INTERFACE I_NodeFactory

METHOD PUBLIC Accept
VAR_INPUT
	Visitor : I_NodeFactoryVisitor;
END_VAR
END_METHOD

METHOD AddNodeAsPrototype : I_NodePrototype
VAR_INPUT
	Path : T_MAXSTRING;
	Node : I_Node;
END_VAR
END_METHOD

METHOD PUBLIC AddNodePrototype
VAR_INPUT
	NodePrototype : I_NodePrototype;
END_VAR
END_METHOD

METHOD PUBLIC InstallNodePack
VAR_INPUT
	NodePack : I_NodePack;
END_VAR
END_METHOD

PROPERTY PUBLIC ABSTRACT NodePrototypes : I_NodePrototypes
GET
END_GET
END_PROPERTY

METHOD PUBLIC TryCreateNodeByType : BOOL
VAR_INPUT
	Path : T_MAXSTRING;
	Destination : REFERENCE TO I_Node;
END_VAR
END_METHOD

END_INTERFACE

(* stored: Version 1.1.0.1, ProductVersion 3.1.4024.12
   Itf I_NodeFactory: Id {1c91137c-0d76-4a0b-982f-ff1013ab557c}
   Method Accept: Id {f6a58bad-0d11-4651-b4e3-e6b638da37c0}
   Method AddNodeAsPrototype: Id {3c290acf-ef58-4296-9f99-efa7638f18a5}
   Method AddNodePrototype: Id {fca90214-0e16-4176-8cb8-b68284861d51}
   Method InstallNodePack: Id {eeb92a5b-c90e-441b-8a57-23a935768eb2}
   Property NodePrototypes: Id {82e304d3-cf5f-4e21-8935-71cbe599f257}
   Get Get: Id {4cb802dd-fdb8-4d8d-8602-1230b292a15c}
   Method TryCreateNodeByType: Id {c6542a73-8c2a-431b-a035-4be5151b15ee} *)
